INTERFACE I_OutputPortChangedEvent extends I_Event

PROPERTY PUBLIC Target : I_OutputPort
GET
END_GET
END_PROPERTY

END_INTERFACE

(* stored: Version 1.1.0.1, ProductVersion 3.1.4024.12
   Itf I_OutputPortChangedEvent: Id {46814cab-cfb9-082d-00e1-321f4992593e}
   Property Target: Id {55d2aa7f-9128-0984-03ce-0c0d27bddc0d}
   Get Get: Id {0b6c7bf7-d71e-065e-344f-795d48ed80c7} *)
